Yaskawa INFORM job: yellow_cover_19_07_23_cylinder_program.JBI

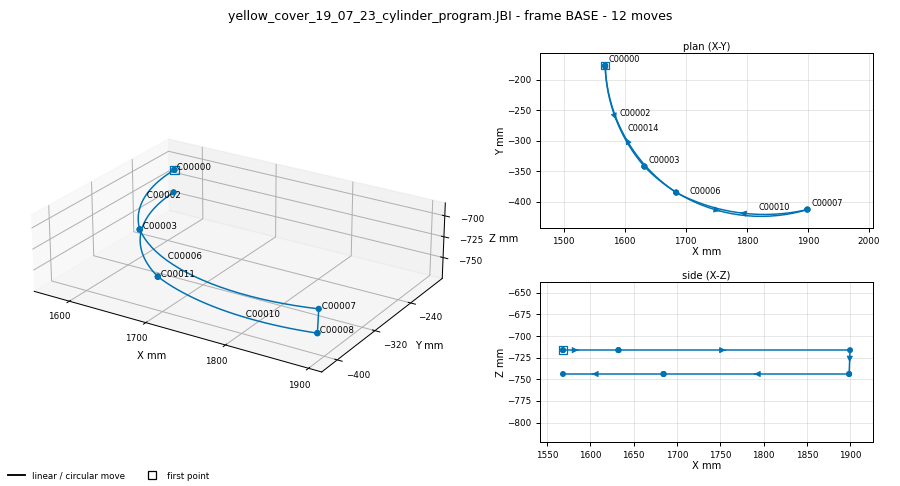
[picture p0: tool path of yellow_cover_19_07_23_cylinder_program.JBI in frame BASE, 12 of 22 moves have a stored position in this frame; points joined in program order, loops and branches not executed]
/JOB
//NAME yellow_cover_19_07_23_cylinder_program
//POS
///NPOS 16,0,16,0,0,0
///TOOL 0
///POSTYPE BASE
///RECTAN
///RCONF 0,0,0,0,0,0,0,0,0,0,0,0,0,0,0,0,0,0,0,0,0,0,0,0
C00000=1568.243225,-177.023699,-716.273960,180.000000,-60.000000,1.663606
C00001=1568.243225,-177.023699,-716.273960,180.000000,-60.000000,1.663606
C00002=1586.144909,-265.752014,-716.273960,180.000000,-60.000000,22.336579
C00003=1632.369762,-342.326442,-716.273960,-180.000000,-60.000000,42.630648
C00004=1632.369762,-342.326442,-716.273960,-180.000000,-60.000000,42.630648
C00005=1632.369762,-342.326442,-716.273960,-180.000000,-60.000000,42.630648
C00006=1699.877891,-393.279600,-716.273960,180.000000,-60.000000,61.774211
C00007=1899.867289,-412.665038,-716.273960,180.000000,-60.000000,108.222941
C00008=1898.828038,-412.861045,-743.842460,-180.000000,-60.000000,107.785455
C00009=1898.828038,-412.861045,-743.842460,-180.000000,-60.000000,107.785455
C00010=1813.763853,-420.437788,-743.842460,180.000000,-60.000000,88.431371
C00011=1684.437246,-384.938188,-743.842460,180.000000,-60.000000,57.740706
C00012=1684.437246,-384.938188,-743.842460,180.000000,-60.000000,57.740706
C00013=1684.437246,-384.938188,-743.842460,180.000000,-60.000000,57.740706
C00014=1598.329194,-289.773211,-743.842460,180.000000,-60.000000,28.485396
C00015=1568.259982,-179.239344,-743.842460,-180.000000,-60.000000,2.291810
///POSTYPE PULSE
///PULSE
EX00000=0
EX00001=92160
EX00002=184320
EX00003=276480
///POSTYPE PULSE
///PULSE
EC00000=0
EC00001=0
EC00002=0
EC00003=0
EC00004=0
EC00005=0
EC00006=0
EC00007=0
EC00008=0
EC00009=0
EC00010=0
EC00011=0
EC00012=0
EC00013=0
EC00014=0
EC00015=0
//INST
///DATE 2023/08/07 14:38
///ATTR SC,RW,RJ
////FRAME BASE
///GROUP1 RB1,ST1
NOP
MOVJ P009 EX000 VJ=15.00
MOVJ P009 VJ=15.00
MOVJ C00000 EC00000 VJ=15.0
CALL JOB:SPYON
MOVC C00001 EC00001 V=150.0
MOVC C00002 EC00002 V=150.0
MOVC C00003 EC00003 V=150.0
MOVL C00004 EC00004 V=150.0
MOVC C00005 EC00005 V=150.0
MOVC C00006 EC00006 V=150.0
MOVC C00007 EC00007 V=150.0
MOVL C00008 EC00008 V=150.0
MOVC C00009 EC00009 V=150.0
MOVC C00010 EC00010 V=150.0
MOVC C00011 EC00011 V=150.0
MOVL C00012 EC00012 V=150.0
MOVC C00013 EC00013 V=150.0
MOVC C00014 EC00014 V=150.0
MOVC C00015 EC00015 V=150.0
CALL JOB:SPYOF
MOVJ P009 VJ=15.00
MOVJ P009 VJ=15.00
MOVJ P009 VJ=15.00
MOVJ P009 VJ=15.00
END
